# B&R Automation Studio project Laba_1
Automation Studio 4.5.2.102

## Configuration Config1

### Task classes (Cpu.sw)
```
Cyclic#4:
  Program1 <- Program1.prg
Libraries: Motor
```

### Hardware
```
4PP065_0571_P74 : 4PP065.0571-P74 v1.1.2.0
  Connector IF5:
    ActivateDevice = 1
  ConfigurationID = laba1_Config1
  Simulation = 1
```

## Logical view

Binary libraries used (declarations not repeated): operator, runtime, astime, AsIecCon

### Package Logical/Libraries - Global libraries

### Library Logical/Libraries/Motor (ANSIC)

#### Motor.fun - Exported functions and function blocks
```iecst
{REDUND_ERROR} FUNCTION_BLOCK FB_Integrator (*TODO: Add your comment here*) (*$GROUP=User,$CAT=User,$GROUPICON=User.png,$CATICON=User.png*)
	VAR_INPUT
		in : REAL;
	END_VAR
	VAR_OUTPUT
		out : {REDUND_UNREPLICABLE} REAL;
	END_VAR
	VAR
		dt : REAL;
	END_VAR
END_FUNCTION_BLOCK

{REDUND_ERROR} FUNCTION_BLOCK FB_Motor (*TODO: Add your comment here*) (*$GROUP=User,$CAT=User,$GROUPICON=User.png,$CATICON=User.png*)
	VAR_INPUT
		u : REAL;
	END_VAR
	VAR_OUTPUT
		w : {REDUND_UNREPLICABLE} REAL;
		phi : {REDUND_UNREPLICABLE} REAL;
	END_VAR
	VAR
		integrator : FB_Integrator;
		Tm : REAL;
		ke : REAL;
		dt : REAL;
	END_VAR
END_FUNCTION_BLOCK

{REDUND_ERROR} FUNCTION_BLOCK FB_Regulator (*TODO: Add your comment here*) (*$GROUP=User,$CAT=User,$GROUPICON=User.png,$CATICON=User.png*)
	VAR_INPUT
		e : REAL;
	END_VAR
	VAR_OUTPUT
		u : {REDUND_UNREPLICABLE} REAL;
	END_VAR
	VAR
		k_p : REAL;
		k_i : REAL;
		integrator : FB_Integrator;
		iyOld : REAL;
		max_abs_value : REAL;
		e_p : REAL;
		dt : REAL;
	END_VAR
END_FUNCTION_BLOCK
```

#### FB_Integrator.c
```c
#include <bur/plctypes.h>
#ifdef __cplusplus
	extern "C"
	{
#endif
	#include "Motor.h"
#ifdef __cplusplus
	};
#endif
/* TODO: Add your comment here */
void FB_Integrator(struct FB_Integrator* inst)
{
	/*TODO: Add your code here*/
	inst->out += inst->in;
}
```

#### FB_Motor.c
```c
#include <bur/plctypes.h>
#ifdef __cplusplus
	extern "C"
	{
#endif
	#include "Motor.h"
#ifdef __cplusplus
	};
#endif
/* TODO: Add your comment here */
void FB_Motor(struct FB_Motor* inst)
{
	/*TODO: Add your code here*/
	inst->integrator.in = (inst->u / inst->ke - inst->w) * (inst->dt / inst->Tm);
	FB_Integrator(&(inst->integrator));
	inst->w = inst->integrator.out;
	inst->integrator.in = inst->w * inst->dt;
	FB_Integrator(&(inst->integrator));
	inst->phi = inst->integrator.out;
}
```

#### FB_Regulator.c
```c
#include <bur/plctypes.h>
#ifdef __cplusplus
	extern "C"
	{
#endif
	#include "Motor.h"
#ifdef __cplusplus
	};
#endif
/* TODO: Add your comment here */
void FB_Regulator(struct FB_Regulator* inst)
{
	/*TODO: Add your code here*/
	inst->integrator.in = +inst->iyOld + inst->e*inst->k_i*inst->dt;
	FB_Integrator(&(inst->integrator));
	inst->e_p = inst->e * inst->k_p;
	if (inst->e_p>inst->max_abs_value || inst->e_p < -inst->max_abs_value) {
		if (inst->e_p>0) inst->e_p = inst->max_abs_value;
		else inst->e_p = -inst->max_abs_value;
	}
	inst->e_p += inst->integrator.out;
	if (inst->e_p<inst->max_abs_value || inst->e_p > -inst->max_abs_value) inst->u = inst->e_p;
	else
	{
		if (inst->e_p>0) inst->u = inst->max_abs_value;
		else inst->u = -inst->max_abs_value;
	}
	inst->iyOld = inst->u - inst->e_p;
}
```

### Program Logical/Program1 (ANSIC)

#### Main.c - Init, cyclic, exit code
```c
#include <bur/plctypes.h>

#ifdef _DEFAULT_INCLUDES
	#include <AsDefault.h>
#endif

void _INIT ProgramInit(void)
{
	Enable = 1;
	count = 0;
	Speed = 0;

	fb_motor.dt = 0.01;
	fb_motor.ke = 0.24;
	fb_motor.Tm = 0.1;
	fb_motor2.dt = 0.01;
	fb_motor2.ke = 0.24;
	fb_motor2.Tm = 0.1;

	fb_controller.dt = 0.01;
	fb_controller.k_p = 7;
	fb_controller.k_i = 5;
	fb_controller.max_abs_value = 24;
}

void _CYCLIC ProgramCyclic(void)
{
	if(Enable == 1) {
		count += 10;
		if(count >= 400 && count <= 2000) Speed = 40;
		else {
			Speed = 5;
		}
		if(count >= 2000){
			count = 0;
		}
	}
	else Speed = 0;

	fb_controller.e = Speed - fb_motor.w;
	fb_motor2.u = Speed * fb_motor2.ke;
	fb_motor.u = fb_controller.u * fb_motor.ke;
	FB_Regulator(&fb_controller);
	FB_Motor(&fb_motor);
	FB_Motor(&fb_motor2);

}

void _EXIT ProgramExit(void)
{

}
```

#### Variables.var - Local variables
```iecst
VAR
	Enable : BOOL;
	Speed : REAL;
	fb_controller : FB_Regulator;
	fb_motor : FB_Motor;
	fb_motor2 : FB_Motor;
	count : REAL;
	integrator : FB_Integrator;
END_VAR
```

Listed in the project but not available here: Logical/Global.typ, Logical/Global.var, Logical/Libraries/Motor/Types.typ, Logical/Libraries/Motor/Constants.var, Logical/Program1/Types.typ
